TYPE OutputBase_10CEE7DE :
STRUCT
END_STRUCT
END_TYPE

(* stored: Version 1.2.0.0, ProductVersion 3.1.4024.9
   DUT OutputBase_10CEE7DE: Id {8e24bdac-8d4f-4979-ae9c-5afb8a6fef4a} *)
